FUNCTION_BLOCK FB_TestHTTP_Head
VAR_INPUT
	fbClient : REFERENCE TO FB_IotHttpClient;
END_VAR
VAR	
	fbRequest: FB_IotHttpRequest;
	fbJson: FB_JsonDomParser;
	bSend : BOOL;
	bContinuous : BOOL;
	state : UDINT;
	
	RisingEdge		: R_TRIG;	
	sContentLen: STRING(256);	
	
	bJsonRes : BOOL;
	jsonDoc    : SJsonValue;
	jsonVal    : SJsonValue;
		
	reqCount : UDINT;		
	invResCount : UDINT := 0;
	invResValCount : UDINT := 0;
	resVal:STRING;
	nResCnt : UDINT;
	nErrCnt1 : UDINT;
	nErrCnt2 : UDINT;
		
	valOkCount: UDINT;
	
	//http://jsonplaceholder.typicode.com/todos/1
	sUri: STRING(255) := '/posts/1';
	eRequestType : ETcIotHttpRequestType := ETcIotHttpRequestType.HTTP_HEAD;		
END_VAR

RisingEdge( CLK:= bSend );
CASE state OF
0:		
	IF fbClient.bConfigured AND (RisingEdge.Q OR bContinuous) THEN 
		IF fbRequest.SendRequest(sUri:=sUri, fbClient:=fbClient, eRequestType:=eRequestType, 0, 0, 0) THEN				
			state := 1;
			reqCount:=reqCount+1;
		END_IF					
	END_IF
1:
	IF NOT fbRequest.bBusy THEN
			IF NOT fbRequest.bError THEN				 
				IF fbRequest.GetHeaderField('Content-Length', ADR(sContentLen), SIZEOF(sContentLen)) THEN 
					IF STRING_TO_UDINT(sContentLen) = 292 THEN
						valOkCount:=valOkCount+1;
					ELSE
						invResValCount:=invResValCount+1;
					END_IF
				ELSE
					invResCount:=invResCount+1;
				END_IF
			ELSE
				nErrCnt2:=nErrCnt2+1;
			END_IF
			state :=0;				
	END_IF  	
END_CASE
fbClient.Execute();

END_FUNCTION_BLOCK

(* stored: Version 1.1.0.1, ProductVersion 3.1.4024.0
   POU FB_TestHTTP_Head: Id {ea1d8295-f351-4741-a791-0797213049c4}, SpecialFunc None *)
